FUNCTION_BLOCK MockObj IMPLEMENTS I_Cyclic, I_Initialisable, I_Object, I_Resettable
VAR
	_isRegistered : BOOL;
END_VAR

METHOD Cycle : HRESULT
END_METHOD

METHOD Initialise : HRESULT
END_METHOD

{warning 'Add property implementation'}
PROPERTY Initialised : BOOL
GET
END_GET
END_PROPERTY

METHOD IsRegistered : BOOL
VAR_INPUT
END_VAR
IsRegistered := _isRegistered;
END_METHOD

METHOD RegisterWithParent
VAR_INPUT
	Parent	: I_HostObjects;
END_VAR
IF NOT _isRegistered THEN
	IF SUCCEEDED( Parent.RegisterCyclic(THIS^)) AND SUCCEEDED(Parent.RegisterInitialisable(THIS^)) THEN
		_isRegistered := TRUE;
	ELSE
		_isRegistered := FALSE;
	END_IF
END_IF
END_METHOD

METHOD Reset : Base_Library.HRESULT
END_METHOD

END_FUNCTION_BLOCK

(* stored: Version 1.1.0.1
   POU MockObj: Id {459c9319-db86-4d6a-b774-a97d62f0aee0}, SpecialFunc None
   Method Cycle: Id {2fdaa782-1cce-42d3-b0fd-0a553501ea73}
   Method Initialise: Id {b6fb438d-078a-4d9d-ba13-f31f733124cc}
   Property Initialised: Id {9ccefc82-4611-4153-984f-16110f1bc2dd}
   Get Get: Id {704bdb38-63cd-4146-9195-7eb236f2d453}
   Method IsRegistered: Id {432ff809-df19-4dfc-b853-62c50ce79958}
   Method RegisterWithParent: Id {53309e55-7b39-4961-93ff-498d9c30e110}
   Method Reset: Id {fdee9a2d-cec1-4e56-8d77-d56933a1dff5} *)
